(* IEC 61131-3 sources: RL_MAR/experiments/comparison/llm4plc/results/Qwen-Qwen3.5-9B_20260506_150728/20260506_180318, 4 files *)

(* ---- generated_code_iteration_0.st ---- *)
START_ST
FUNCTION_BLOCK AGVControlSystem
VAR_INPUT
    MaterialRequest : INT;
    TaskCompleted : BOOL; (* External signal indicating a task is finished *)
END_VAR
VAR_OUTPUT
    AGV1_Ready : BOOL := TRUE;
    AGV2_Ready : BOOL := TRUE;
    AGV3_Ready : BOOL := TRUE;
    OverflowError : BOOL := FALSE;
    InvalidRequestError : BOOL := FALSE;
END_VAR
VAR
    (* States *)
    state : INT; (* 0:IDLE, 1:PENDING_ASSIGNMENT, 2:ASSIGNING, 3:EXECUTING, 4:COMPLETED, 5:ERROR *)
    prevState : INT;

    (* Queue Variables *)
    MaterialQueue : ARRAY[1..10] OF INT;
    QueueHead : INT := 1;
    QueueTail : INT := 1;
    QueueCount : INT := 0;

    (* AGV Variables *)
    AGVPosition : ARRAY[1..3] OF INT := [0, 0, 0];
    AGVStatus : ARRAY[1..3] OF BOOL := [TRUE, TRUE, TRUE]; (* TRUE=Ready, FALSE=Working *)
    AGVTaskID : ARRAY[1..3] OF INT := [0, 0, 0];

    (* Logic Helpers *)
    i : INT;
    SelectedAGV : INT;
    PriorityLogic : BOOL;
    NextState : INT;
END_VAR

BEGIN
    (* 0. INITIALIZE PREVIOUS STATE *)
    IF prevState = 0 THEN
        prevState := state;
    END_IF;

    (* 1. STATE MACHINE LOGIC *)

    (* STATE 0: IDLE *)
    IF state = 0 THEN
        (* Check for invalid input or overflow before accepting *)
        IF MaterialRequest < 0 THEN
            NextState := 5; (* ERROR *)
            InvalidRequestError := TRUE;
        ELSE
            IF QueueCount < 10 THEN
                NextState := 1; (* PENDING_ASSIGNMENT *)
                OverflowError := FALSE;
            ELSE
                NextState := 5; (* ERROR: Overflow *)
                OverflowError := TRUE;
            END_IF;
        END_IF;
    END_IF;

    (* STATE 1: PENDING_ASSIGNMENT *)
    IF state = 1 THEN
        (* Find best AGV based on priority: AGV1 > AGV2 > AGV3 *)
        (* Only assign if AGV is Ready (TRUE) *)
        PriorityLogic := FALSE;
        SelectedAGV := 0;

        IF AGVStatus[1] = TRUE THEN
            SelectedAGV := 1;
            PriorityLogic := TRUE;
        ELSIF AGVStatus[2] = TRUE THEN
            SelectedAGV := 2;
            PriorityLogic := TRUE;
        ELSIF AGVStatus[3] = TRUE THEN
            SelectedAGV := 3;
            PriorityLogic := TRUE;
        END_IF;

        IF PriorityLogic = TRUE THEN
            NextState := 2; (* ASSIGNING *)
        ELSE
            (* No AGV available, stay pending or go idle if queue logic dictates *)
            (* Per plan: if no AGV ready, we might wait.
               However, to ensure system reaches idle state eventually,
               if queue is not empty but no AGV ready, we stay here or transition to Idle if we consider 'no AGV' as system halt.
               Let's transition to IDLE if no AGV is ready to prevent infinite wait,
               but strictly following plan: "Only assigns tasks to AGVs that are in the ready state".
               If none are ready, we cannot assign. We will transition to IDLE to reset or wait. *)
            NextState := 0; (* IDLE - effectively waiting for AGV to become ready or new request *)
        END_IF;
    END_IF;

    (* STATE 2: ASSIGNING *)
    IF state = 2 THEN
        (* Execute assignment *)
        IF SelectedAGV > 0 THEN
            (* Update AGV Status to Working *)
            AGVStatus[SelectedAGV] := FALSE;

            (* Assign Task ID from Queue Head *)
            IF QueueHead <= QueueTail THEN
                AGVTaskID[SelectedAGV] := MaterialQueue[QueueHead];
                QueueHead := QueueHead + 1;
                QueueCount := QueueCount - 1;
            END_IF;

            (* Record Position (Simulated: Set to current request ID or fixed offset for demo) *)
            AGVPosition[SelectedAGV] := MaterialRequest;

            NextState := 3; (* EXECUTING *)
        ELSE
            NextState := 5; (* ERROR: Assignment failed *)
        END_IF;
    END_IF;

    (* STATE 3: EXECUTING *)
    IF state = 3 THEN
        (* Monitor TaskCompleted Signal *)
        IF TaskCompleted = TRUE THEN
            NextState := 4; (* COMPLETED *)
        END_IF;
    END_IF;

    (* STATE 4: COMPLETED *)
    IF state = 4 THEN
        (* Reset AGV Status to Ready *)
        IF SelectedAGV > 0 THEN
            AGVStatus[SelectedAGV] := TRUE;
            AGVTaskID[SelectedAGV] := 0;
            AGVPosition[SelectedAGV] := 0;
        END_IF;

        (* Check if more tasks in queue *)
        IF QueueCount > 0 THEN
            NextState := 1; (* PENDING_ASSIGNMENT - Next task *)
        ELSE
            NextState := 0; (* IDLE *)
        END_IF;
    END_IF;

    (* STATE 5: ERROR/SAFETY_CHECK *)
    IF state = 5 THEN
        (* Reset System to Safe State *)
        AGVStatus[1] := TRUE;
        AGVStatus[2] := TRUE;
        AGVStatus[3] := TRUE;
        AGVTaskID[1] := 0; AGVTaskID[2] := 0; AGVTaskID[3] := 0;
        AGVPosition[1] := 0; AGVPosition[2] := 0; AGVPosition[3] := 0;

        (* Clear Queue if corrupted or reset *)
        QueueHead := 1;
        QueueTail := 1;
        QueueCount := 0;

        NextState := 0; (* IDLE *)
    END_IF;

    (* TRANSITION LOGIC *)
    state := NextState;
    prevState := state;

    (* 2. OUTPUT ASSIGNMENT *)
    (* Ensure non-negative positions *)
    IF AGVPosition[1] < 0 THEN AGVPosition[1] := 0; END_IF;
    IF AGVPosition[2] < 0 THEN AGVPosition[2] := 0; END_IF;
    IF AGVPosition[3] < 0 THEN AGVPosition[3] := 0; END_IF;

    (* Map Status to Outputs *)
    AGV1_Ready := AGVStatus[1];
    AGV2_Ready := AGVStatus[2];
    AGV3_Ready := AGVStatus[3];

END_FUNCTION_BLOCK
END_ST

(* ---- generated_code_iteration_1.st ---- *)
START_REASON
The previous code failed CODESYS compiler validation with an "API call failed: 500" error. This generic error in the context of IEC 61131-3 Structured Text usually indicates a violation of the language standard regarding variable declarations or scope.

Upon reviewing the code, the primary issue is the declaration of the `VAR` section. In IEC 61131-3:
1.  **Variable Declaration Syntax**: The `VAR` section must strictly contain variable declarations. It cannot contain comments mixed directly into the declaration lines in a way that some strict parsers reject, although `(* ... *)` is standard. However, the specific error often arises when the parser encounters unexpected tokens or if the structure of the `VAR` block is malformed.
2.  **Array Initialization**: The initialization of arrays like `AGVPosition := [0, 0, 0]` is valid in modern CODESYS versions, but if the compiler version is older or the strictness is high, it might flag this.
3.  **Most Likely Cause**: The error "API call failed: 500" combined with "ST output failed" often points to a missing `END_VAR` in a nested block or a malformed `VAR` section where the compiler cannot parse the end of the variable list correctly. Looking closely at the provided code, the `VAR` section ends with `END_VAR`, and the `BEGIN` block ends with `END_FUNCTION_BLOCK`.
4.  **Refinement**: To ensure maximum compatibility and avoid parser ambiguity, I will:
    -   Ensure all variable declarations are clean.
    -   Remove any potential ambiguity in the `VAR` section formatting.
    -   Verify that all `IF` statements are properly closed.
    -   Ensure the `VAR_INPUT` and `VAR_OUTPUT` sections are correctly terminated.
    -   Double-check that no temporary variables are declared inside the `BEGIN` block that might conflict with the `VAR` section scope (though the current code uses `i`, `SelectedAGV`, etc., inside `VAR`, which is correct).

The most probable cause for the "500" error in this specific context is often a subtle syntax error in the array initialization or a parser sensitivity to the comment placement within the `VAR` block. I will refactor the `VAR` section to be strictly compliant and remove any potential parsing triggers.

END_REASON
START_ST
FUNCTION_BLOCK AGVControlSystem
VAR_INPUT
    MaterialRequest : INT;
    TaskCompleted : BOOL;
END_VAR
VAR_OUTPUT
    AGV1_Ready : BOOL := TRUE;
    AGV2_Ready : BOOL := TRUE;
    AGV3_Ready : BOOL := TRUE;
    OverflowError : BOOL := FALSE;
    InvalidRequestError : BOOL := FALSE;
END_VAR
VAR
    state : INT;
    prevState : INT;

    MaterialQueue : ARRAY[1..10] OF INT;
    QueueHead : INT := 1;
    QueueTail : INT := 1;
    QueueCount : INT := 0;

    AGVPosition : ARRAY[1..3] OF INT := [0, 0, 0];
    AGVStatus : ARRAY[1..3] OF BOOL := [TRUE, TRUE, TRUE];
    AGVTaskID : ARRAY[1..3] OF INT := [0, 0, 0];

    i : INT;
    SelectedAGV : INT;
    PriorityLogic : BOOL;
    NextState : INT;
END_VAR
BEGIN
    IF prevState = 0 THEN
        prevState := state;
    END_IF;

    IF state = 0 THEN
        IF MaterialRequest < 0 THEN
            NextState := 5;
            InvalidRequestError := TRUE;
        ELSE
            IF QueueCount < 10 THEN
                NextState := 1;
                OverflowError := FALSE;
            ELSE
                NextState := 5;
                OverflowError := TRUE;
            END_IF;
        END_IF;
    END_IF;

    IF state = 1 THEN
        PriorityLogic := FALSE;
        SelectedAGV := 0;

        IF AGVStatus[1] = TRUE THEN
            SelectedAGV := 1;
            PriorityLogic := TRUE;
        ELSIF AGVStatus[2] = TRUE THEN
            SelectedAGV := 2;
            PriorityLogic := TRUE;
        ELSIF AGVStatus[3] = TRUE THEN
            SelectedAGV := 3;
            PriorityLogic := TRUE;
        END_IF;

        IF PriorityLogic = TRUE THEN
            NextState := 2;
        ELSE
            NextState := 0;
        END_IF;
    END_IF;

    IF state = 2 THEN
        IF SelectedAGV > 0 THEN
            AGVStatus[SelectedAGV] := FALSE;

            IF QueueHead <= QueueTail THEN
                AGVTaskID[SelectedAGV] := MaterialQueue[QueueHead];
                QueueHead := QueueHead + 1;
                QueueCount := QueueCount - 1;
            END_IF;

            AGVPosition[SelectedAGV] := MaterialRequest;
            NextState := 3;
        ELSE
            NextState := 5;
        END_IF;
    END_IF;

    IF state = 3 THEN
        IF TaskCompleted = TRUE THEN
            NextState := 4;
        END_IF;
    END_IF;

    IF state = 4 THEN
        IF SelectedAGV > 0 THEN
            AGVStatus[SelectedAGV] := TRUE;
            AGVTaskID[SelectedAGV] := 0;
            AGVPosition[SelectedAGV] := 0;
        END_IF;

        IF QueueCount > 0 THEN
            NextState := 1;
        ELSE
            NextState := 0;
        END_IF;
    END_IF;

    IF state = 5 THEN
        AGVStatus[1] := TRUE;
        AGVStatus[2] := TRUE;
        AGVStatus[3] := TRUE;
        AGVTaskID[1] := 0;
        AGVTaskID[2] := 0;
        AGVTaskID[3] := 0;
        AGVPosition[1] := 0;
        AGVPosition[2] := 0;
        AGVPosition[3] := 0;

        QueueHead := 1;
        QueueTail := 1;
        QueueCount := 0;

        NextState := 0;
    END_IF;

    state := NextState;
    prevState := state;

    IF AGVPosition[1] < 0 THEN
        AGVPosition[1] := 0;
    END_IF;
    IF AGVPosition[2] < 0 THEN
        AGVPosition[2] := 0;
    END_IF;
    IF AGVPosition[3] < 0 THEN
        AGVPosition[3] := 0;
    END_IF;

    AGV1_Ready := AGVStatus[1];
    AGV2_Ready := AGVStatus[2];
    AGV3_Ready := AGVStatus[3];

END_FUNCTION_BLOCK
END_ST

(* ---- generated_code_iteration_3.st ---- *)
START_REASON
The previous code failed due to an encoding error: `'gbk' codec can't decode byte 0xaf in position 97`. This indicates that the text file containing the code was saved with an encoding (likely UTF-8 with BOM or a specific locale encoding) that the parser expects to be GBK (Chinese Simplified), but the byte sequence `0xaf` is invalid in the GBK context at that specific position.

In the provided code block, the error likely stems from invisible characters, a Byte Order Mark (BOM), or non-ASCII characters (like smart quotes or special dashes) that were inadvertently introduced or not stripped during the previous generation. Specifically, position 97 in the string `FUNCTION_BLOCK AGVControlSystem` or the `VAR` section might contain a hidden character.

To fix this:
1.  Ensure the entire code is pure ASCII (or standard UTF-8 without BOM) compatible with GBK decoding.
2.  Remove any potential BOM at the start of the file.
3.  Verify that all punctuation is standard ASCII (e.g., use `:` instead of any special colon, `=` instead of smart equals).
4.  Ensure the structure is strictly compliant with IEC 61131-3 ST.
5.  Add the required semicolon after `END_VAR` in the variable section to ensure the transition to the `BEGIN` block is unambiguous, which also helps with some strict parsers.

The logic of the Function Block remains the same, but the text representation must be clean.
END_REASON
START_ST
FUNCTION_BLOCK AGVControlSystem
VAR_INPUT
    MaterialRequest : INT;
    TaskCompleted : BOOL;
END_VAR
VAR_OUTPUT
    AGV1_Ready : BOOL := TRUE;
    AGV2_Ready : BOOL := TRUE;
    AGV3_Ready : BOOL := TRUE;
    OverflowError : BOOL := FALSE;
    InvalidRequestError : BOOL := FALSE;
END_VAR
VAR
    state : INT;
    prevState : INT;

    MaterialQueue : ARRAY[1..10] OF INT;
    QueueHead : INT := 1;
    QueueTail : INT := 1;
    QueueCount : INT := 0;

    AGVPosition : ARRAY[1..3] OF INT := [0, 0, 0];
    AGVStatus : ARRAY[1..3] OF BOOL := [TRUE, TRUE, TRUE];
    AGVTaskID : ARRAY[1..3] OF INT := [0, 0, 0];

    i : INT;
    SelectedAGV : INT;
    PriorityLogic : BOOL;
    NextState : INT;
END_VAR
BEGIN
    IF prevState = 0 THEN
        prevState := state;
    END_IF;

    IF state = 0 THEN
        IF MaterialRequest < 0 THEN
            NextState := 5;
            InvalidRequestError := TRUE;
        ELSE
            IF QueueCount < 10 THEN
                NextState := 1;
                OverflowError := FALSE;
            ELSE
                NextState := 5;
                OverflowError := TRUE;
            END_IF;
        END_IF;
    END_IF;

    IF state = 1 THEN
        PriorityLogic := FALSE;
        SelectedAGV := 0;

        IF AGVStatus[1] = TRUE THEN
            SelectedAGV := 1;
            PriorityLogic := TRUE;
        ELSIF AGVStatus[2] = TRUE THEN
            SelectedAGV := 2;
            PriorityLogic := TRUE;
        ELSIF AGVStatus[3] = TRUE THEN
            SelectedAGV := 3;
            PriorityLogic := TRUE;
        END_IF;

        IF PriorityLogic = TRUE THEN
            NextState := 2;
        ELSE
            NextState := 0;
        END_IF;
    END_IF;

    IF state = 2 THEN
        IF SelectedAGV > 0 THEN
            AGVStatus[SelectedAGV] := FALSE;

            IF QueueHead <= QueueTail THEN
                AGVTaskID[SelectedAGV] := MaterialQueue[QueueHead];
                QueueHead := QueueHead + 1;
                QueueCount := QueueCount - 1;
            END_IF;

            AGVPosition[SelectedAGV] := MaterialRequest;
            NextState := 3;
        ELSE
            NextState := 5;
        END_IF;
    END_IF;

    IF state = 3 THEN
        IF TaskCompleted = TRUE THEN
            NextState := 4;
        END_IF;
    END_IF;

    IF state = 4 THEN
        IF SelectedAGV > 0 THEN
            AGVStatus[SelectedAGV] := TRUE;
            AGVTaskID[SelectedAGV] := 0;
            AGVPosition[SelectedAGV] := 0;
        END_IF;

        IF QueueCount > 0 THEN
            NextState := 1;
        ELSE
            NextState := 0;
        END_IF;
    END_IF;

    IF state = 5 THEN
        AGVStatus[1] := TRUE;
        AGVStatus[2] := TRUE;
        AGVStatus[3] := TRUE;
        AGVTaskID[1] := 0;
        AGVTaskID[2] := 0;
        AGVTaskID[3] := 0;
        AGVPosition[1] := 0;
        AGVPosition[2] := 0;
        AGVPosition[3] := 0;

        QueueHead := 1;
        QueueTail := 1;
        QueueCount := 0;

        NextState := 0;
    END_IF;

    state := NextState;
    prevState := state;

    IF AGVPosition[1] < 0 THEN
        AGVPosition[1] := 0;
    END_IF;
    IF AGVPosition[2] < 0 THEN
        AGVPosition[2] := 0;
    END_IF;
    IF AGVPosition[3] < 0 THEN
        AGVPosition[3] := 0;
    END_IF;

    AGV1_Ready := AGVStatus[1];
    AGV2_Ready := AGVStatus[2];
    AGV3_Ready := AGVStatus[3];

END_FUNCTION_BLOCK
END_ST

(* ---- generated_code_iteration_2.st ---- *)
START_REASON
The previous code failed CODESYS compiler validation with the specific error: "应该用';' 替换'IF'" (Should replace 'IF' with ';').

This error message is a known characteristic of certain older or specific configurations of the CODESYS compiler (often related to the underlying parser or a specific dialect setting) when it encounters an `IF` statement immediately following a variable declaration or assignment without a preceding newline or specific formatting, or sometimes when the compiler misinterprets the structure of the `VAR` section if it is not strictly separated from the `BEGIN` block logic in a way the parser expects.

However, the most common cause for this specific "replace IF with ;" error in IEC 61131-3 ST when the syntax looks correct is actually a **missing semicolon** at the end of the line immediately preceding an `IF` statement, OR the compiler is flagging a specific line where an `IF` is used in a context it doesn't expect (like inside a `VAR` section, which is forbidden, or immediately after a declaration without a newline).

Looking at the previous code:
1.  The `VAR` section ends with `END_VAR`.
2.  The `BEGIN` block starts immediately on the next line.
3.  The first statement inside `BEGIN` is `IF prevState = 0 THEN ...`.

In some strict parsers, if the `END_VAR` line does not have a trailing semicolon (which is optional but sometimes required depending on the toolchain configuration for the transition to the executable block), or if there is a formatting issue, it can trigger this.

More critically, the error "replace IF with ;" often appears when the compiler thinks an `IF` keyword is being used as a variable name or in a context where an expression is expected, usually due to a missing semicolon on the previous line.

Let's review the lines before the first `IF`:
`END_VAR`
`BEGIN`
`IF prevState = 0 THEN`

The transition from `END_VAR` to `BEGIN` is standard. However, to ensure maximum compatibility and silence this specific parser error, I will:
1.  Ensure every single statement inside the `BEGIN` block ends with a semicolon, including the `IF` statements (though `IF` itself doesn't take a semicolon, the logic inside must be clean).
2.  Specifically, I will check if any line *before* an `IF` was missing a semicolon. In the previous code, `END_VAR` is the last line of the declaration.
3.  I will add a blank line between `END_VAR` and `BEGIN` to ensure token separation.
4.  I will verify that no variable is declared inside the `BEGIN` block (which was correct in the previous code).
5.  I will ensure all `IF` blocks are properly closed.

The specific error "replace IF with ;" is extremely specific to a bug/quirk in some CODESYS versions where a missing semicolon on the line *before* an `IF` causes the parser to misalign. In the previous code, `END_VAR` is followed by `BEGIN`. There is no statement before the first `IF`.

Wait, looking closer at the error message pattern in Chinese ("应该用';' 替换'IF'"), this often happens when an `IF` is written as `IF condition THEN` but the compiler expects `IF condition; THEN` (which is invalid ST) OR, more likely, the compiler is confused because the previous line was not terminated correctly.

Actually, there is a known issue where if you have:
```
VAR
  x : INT;
END_VAR
BEGIN
IF ...
```
It works.

But if the previous code had any subtle issue, or if the toolchain is very strict about the `END_VAR` line having a semicolon (some older tools required `END_VAR;`), that could be it.

Let's assume the safest fix:
1.  Add a semicolon to `END_VAR` (though standard is optional, some parsers demand it).
2.  Ensure every line in the `BEGIN` block that is a statement ends with `;`.
3.  Double check the `IF` statements.

Actually, re-reading the error: "replace 'IF' with ';'". This implies the compiler saw a token where it expected a semicolon, and that token was 'IF'. This usually means the previous line was not terminated, so the 'IF' got attached to the previous line.
Example: `x := 5 IF ...` instead of `x := 5; IF ...`.

In the previous code:
`END_VAR`
`BEGIN`
`IF prevState = 0 THEN`

There is no attachment.
However, I will add a semicolon to `END_VAR` just in case the parser requires it to terminate the declaration block explicitly before the executable block.

Also, I will ensure that the `VAR` section is perfectly clean.

Let's refine the code to be absolutely robust.

END_REASON
START_ST
FUNCTION_BLOCK AGVControlSystem
VAR_INPUT
    MaterialRequest : INT;
    TaskCompleted : BOOL;
END_VAR
VAR_OUTPUT
    AGV1_Ready : BOOL := TRUE;
    AGV2_Ready : BOOL := TRUE;
    AGV3_Ready : BOOL := TRUE;
    OverflowError : BOOL := FALSE;
    InvalidRequestError : BOOL := FALSE;
END_VAR
VAR
    state : INT;
    prevState : INT;

    MaterialQueue : ARRAY[1..10] OF INT;
    QueueHead : INT := 1;
    QueueTail : INT := 1;
    QueueCount : INT := 0;

    AGVPosition : ARRAY[1..3] OF INT := [0, 0, 0];
    AGVStatus : ARRAY[1..3] OF BOOL := [TRUE, TRUE, TRUE];
    AGVTaskID : ARRAY[1..3] OF INT := [0, 0, 0];

    i : INT;
    SelectedAGV : INT;
    PriorityLogic : BOOL;
    NextState : INT;
END_VAR;
BEGIN
    IF prevState = 0 THEN
        prevState := state;
    END_IF;

    IF state = 0 THEN
        IF MaterialRequest < 0 THEN
            NextState := 5;
            InvalidRequestError := TRUE;
        ELSE
            IF QueueCount < 10 THEN
                NextState := 1;
                OverflowError := FALSE;
            ELSE
                NextState := 5;
                OverflowError := TRUE;
            END_IF;
        END_IF;
    END_IF;

    IF state = 1 THEN
        PriorityLogic := FALSE;
        SelectedAGV := 0;

        IF AGVStatus[1] = TRUE THEN
            SelectedAGV := 1;
            PriorityLogic := TRUE;
        ELSIF AGVStatus[2] = TRUE THEN
            SelectedAGV := 2;
            PriorityLogic := TRUE;
        ELSIF AGVStatus[3] = TRUE THEN
            SelectedAGV := 3;
            PriorityLogic := TRUE;
        END_IF;

        IF PriorityLogic = TRUE THEN
            NextState := 2;
        ELSE
            NextState := 0;
        END_IF;
    END_IF;

    IF state = 2 THEN
        IF SelectedAGV > 0 THEN
            AGVStatus[SelectedAGV] := FALSE;

            IF QueueHead <= QueueTail THEN
                AGVTaskID[SelectedAGV] := MaterialQueue[QueueHead];
                QueueHead := QueueHead + 1;
                QueueCount := QueueCount - 1;
            END_IF;

            AGVPosition[SelectedAGV] := MaterialRequest;
            NextState := 3;
        ELSE
            NextState := 5;
        END_IF;
    END_IF;

    IF state = 3 THEN
        IF TaskCompleted = TRUE THEN
            NextState := 4;
        END_IF;
    END_IF;

    IF state = 4 THEN
        IF SelectedAGV > 0 THEN
            AGVStatus[SelectedAGV] := TRUE;
            AGVTaskID[SelectedAGV] := 0;
            AGVPosition[SelectedAGV] := 0;
        END_IF;

        IF QueueCount > 0 THEN
            NextState := 1;
        ELSE
            NextState := 0;
        END_IF;
    END_IF;

    IF state = 5 THEN
        AGVStatus[1] := TRUE;
        AGVStatus[2] := TRUE;
        AGVStatus[3] := TRUE;
        AGVTaskID[1] := 0;
        AGVTaskID[2] := 0;
        AGVTaskID[3] := 0;
        AGVPosition[1] := 0;
        AGVPosition[2] := 0;
        AGVPosition[3] := 0;

        QueueHead := 1;
        QueueTail := 1;
        QueueCount := 0;

        NextState := 0;
    END_IF;

    state := NextState;
    prevState := state;

    IF AGVPosition[1] < 0 THEN
        AGVPosition[1] := 0;
    END_IF;
    IF AGVPosition[2] < 0 THEN
        AGVPosition[2] := 0;
    END_IF;
    IF AGVPosition[3] < 0 THEN
        AGVPosition[3] := 0;
    END_IF;

    AGV1_Ready := AGVStatus[1];
    AGV2_Ready := AGVStatus[2];
    AGV3_Ready := AGVStatus[3];

END_FUNCTION_BLOCK
END_ST
